FUNCTION GetLeadingSegmentFromNamespace : T_MAXSTRING
VAR_INPUT
	Symbol : T_MAXSTRING;
END_VAR
VAR
    splitSymbol : T_MAXSTRING;
END_VAR

FindAndSplitChar( 
	sSeparatorChar := '.',  
	pSrcString := ADR(Symbol),                                  
	pLeftString := ADR(GetLeadingSegmentFromNamespace),   
	nLeftSize := SIZEOF(GetLeadingSegmentFromNamespace),                                  
	pRightString := ADR(splitSymbol), 
	nRightSize := SIZEOF(splitSymbol),                                
	bSearchFromRight := FALSE 
);

END_FUNCTION

(* stored: Version 1.1.0.1, ProductVersion 3.1.4024.12
   POU GetLeadingSegmentFromNamespace: Id {0c1c3bd0-cc69-056c-3f81-bb619e60ddc4}, SpecialFunc None *)
